Fanuc KAREL source: kb00168.KL

-- PROVISIONAL review KL for V1013-1; original PC SHA256 f4b49357302cd392e17eeee60a60e3f24c47c792e5df4c4cd619d5b43de6b708
-- Incomplete behavior may be omitted. Consult companion uncertainty JSON. Do not deploy.
PROGRAM KB00168
%NOLOCKGROUP
BEGIN
  -- UNRESOLVED_PC offsets 5-14; opcodes 3F,75
  -- UNRESOLVED_PC offsets 19-26; opcodes 9D,23
  -- UNRESOLVED_PC offsets 31-49; opcodes 27,22,2A,22,31
  -- UNRESOLVED_PC offsets 54-58; opcodes 7F
END KB00168
